// Base function block for collections.
{attribute 'enable_dynamic_creation'}
{attribute 'no_explicit_call' := 'direct call for this function block is not allowed'}
FUNCTION_BLOCK ABSTRACT FB_Collection IMPLEMENTS I_Collection
VAR
	Count : T_Capacity;
	Error : T_Error := F_Error(0,0,'');
END_VAR

// Number of items in the collection.
PROPERTY _Count : T_Capacity
GET
_Count := THIS^.Count;
END_GET
SET // PROTECTED
THIS^.Count := _Count;
END_SET
END_PROPERTY

// Error status of the collection.
PROPERTY _Error_Status : T_Error
GET
_Error_Status := THIS^.Error;
END_GET
SET // PROTECTED
THIS^.Error := _Error_Status;
END_SET
END_PROPERTY

// Checks if collection is empty.
PROPERTY _Is_Empty : BOOL
GET
_Is_Empty := THIS^._Count <= 0;
END_GET
END_PROPERTY

METHOD PROTECTED Clear_Error
VAR_INPUT
END_VAR
THIS^._Error_Status := F_Error(0,0,'');
END_METHOD

// Decrement collection count by 1.
METHOD PROTECTED Decrement_Count
THIS^._Count := THIS^._Count - 1;
END_METHOD

// Increments collection count by 1
METHOD PROTECTED Increment_Count
VAR_INPUT
END_VAR
THIS^._Count := THIS^._Count + 1;
END_METHOD

END_FUNCTION_BLOCK

(* stored: Version 1.1.0.1, ProductVersion 3.1.4024.4
   POU FB_Collection: Id {3c9ea3d8-ae44-47bf-9b7d-af564525410b}, SpecialFunc None
   Folder Protected: Id {acdb10a6-986b-4745-9dbe-96d7b34d0af6}
   Property _Count: Id {8abb8e9e-5743-493b-8b6b-ae6ae38b4c23}
   Get Get: Id {b2897a6b-3882-4669-8cdd-c032ba488ee5}
   Set Set: Id {ebc8b79d-0403-4cb0-af57-ea568b7a36bb}
   Property _Error_Status: Id {84873416-64cd-47b2-af34-a6a695821f58}
   Get Get: Id {e71ab532-eaba-418e-ad7c-71d8b88aa1f1}
   Set Set: Id {275452ae-7b92-4d51-acad-ec1f0a18b315}
   Property _Is_Empty: Id {872db091-b113-44bc-b405-6204d5a476a8}
   Get Get: Id {f9e47430-4ea0-4423-8059-4036f26f7e46}
   Method Clear_Error: Id {e93b111a-9491-4696-9fb2-6330c84a0c7e}
   Method Decrement_Count: Id {93b785e8-52d9-4b0a-9a50-f3b0e6dc1051}
   Method Increment_Count: Id {1950e653-7dd1-4b1e-9eb2-3fa3b0d306c6} *)
